// TIA Portal V20 export
ORGANIZATION_BLOCK "Main"   // OB1, LAD, ProgramCycle
TITLE = Main Program Sweep (Cycle)
{ S7_Optimized_Access := 'TRUE' }
// stored: SetENOAutomatically false
   VAR_INPUT
      Initial_Call : Bool;
      Remanence : Bool;
   END_VAR
BEGIN

REGION Network 1: IO Apply
   // Call FC_IO_Apply
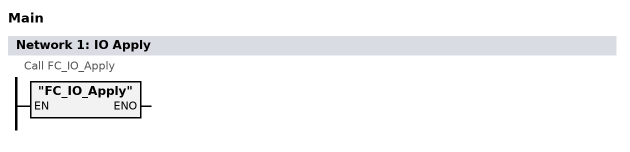
   RUNG wire#powerrail
      "FC_IO_Apply"()
   END_RUNG
   // the same network as SCL:
   "FC_IO_Apply"();
END_REGION
END_ORGANIZATION_BLOCK
